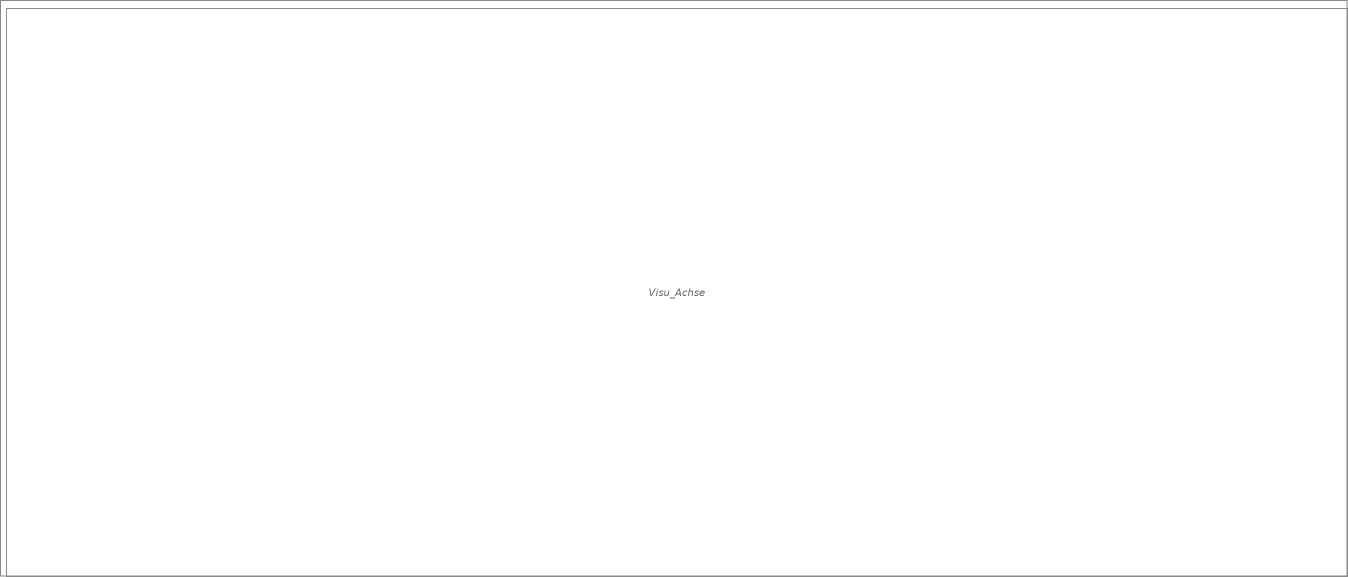
VISUALIZATION Achse_R  // 1348x577
    Frame (6,8 1342x569)
        shows Visu_Achse(Axis := MAIN.Axis_R)
END_VISUALIZATION

(* stored: Version 1.1.0.1, ProductVersion 3.1.4024.12
   Visu Achse_R: Id {8dee067a-d472-41b1-bacb-eff41e1324ae} *)
